{attribute 'qualified_only'}
{attribute 'strict'}
TYPE E_GripperState :
(
	Undefined,
	Open,
	HalfClosed,
	FullyClosed
)USINT;
END_TYPE

(* stored: Version 1.1.0.1, ProductVersion 3.1.4024.11
   DUT E_GripperState: Id {9d1a48ed-8200-4b11-8800-37c33315d570} *)
